// TwinCAT 3 PLC project TcPluginFramework
// Title: TcPluginFramework
// Company: Loupe
// ProjectVersion: 1.0.0
// ProgramVersion: 3.1.4024.0
// libraries:
//   Tc2_System, * (Beckhoff Automation GmbH)
//   TcUnit, * (www.tcunit.org)
// project tree:
//   DUTs/ ComponentBaseInternal.TcDUT, TaskBaseInternal.TcDUT
//   GVLs/ GVLPluginFramework.TcGVL
//   Interfaces/ IPlugin.TcIO, IPluginRunner.TcIO, ITaskState.TcIO
//   POUs/ ComponentBase.TcPOU, LogMessage.TcPOU, PluginRunner.TcPOU, TaskBase.TcPOU
//   Test/ TaskBaseExtended.TcPOU, TESTPRG.TcPOU

// ---- DUTs/ComponentBaseInternal.TcDUT
TYPE
    ComponentBaseInternal :
    STRUCT
        _initDone : BOOL;
        _ready : BOOL;
        _plugins : PluginRunner;
    END_STRUCT
END_TYPE

// ---- DUTs/TaskBaseInternal.TcDUT
TYPE
    TaskBaseInternal :
    STRUCT
        _state : UDINT;
        _newCommand : BOOL;
    END_STRUCT
END_TYPE

// ---- GVLs/GVLPluginFramework.TcGVL
{attribute 'qualified_only'}
VAR_GLOBAL
END_VAR
VAR_GLOBAL CONSTANT
	MAX_NUM_PLUGIN_RUNNERS: USINT := 20;
	MAI_NUM_PLUGIN_RUNNERS: USINT := MAX_NUM_PLUGIN_RUNNERS - 1;
END_VAR
VAR_GLOBAL
    LogLevel : INT;
END_VAR

// ---- Interfaces/IPlugin.TcIO
// Copyright (c) 2024 Loupe (https://loupe.team), provided under the MIT License.

INTERFACE IPlugin EXTENDS __SYSTEM.IQueryInterface

METHOD Run : BOOL
VAR_INPUT
END_VAR
END_METHOD

END_INTERFACE

// ---- Interfaces/IPluginRunner.TcIO
// Copyright (c) 2024 Loupe (https://loupe.team), provided under the MIT License.

INTERFACE IPluginRunner EXTENDS __System.IQueryInterface

METHOD RegisterPlugin
VAR_INPUT
    plugin : IPlugin;
END_VAR
END_METHOD

END_INTERFACE

// ---- Interfaces/ITaskState.TcIO
// Copyright (c) 2024 Loupe (https://loupe.team), provided under the MIT License.

INTERFACE ITaskState

METHOD Cyclic : BOOL
END_METHOD

METHOD Inihibits : BOOL
VAR_INPUT
END_VAR
END_METHOD

METHOD NewCommandState : BOOL
VAR_INPUT
    newTaskState : ENUM;
END_VAR
END_METHOD

PROPERTY NewTaskCommand : BOOL
GET
END_GET
END_PROPERTY

METHOD StateErrored : BOOL
VAR_INPUT
END_VAR
END_METHOD

METHOD StateFinished : BOOL
VAR_INPUT
END_VAR
END_METHOD

METHOD StateMachine : BOOL
VAR_INPUT
END_VAR
END_METHOD

{attribute 'monitoring' := 'call'}
PROPERTY TaskReady : Bool
GET
END_GET
SET
END_SET
END_PROPERTY

{attribute 'monitoring' := 'call'}
PROPERTY TaskState : ENUM
GET
END_GET
END_PROPERTY

METHOD UpdateState : BOOL
VAR_INPUT
END_VAR
END_METHOD

END_INTERFACE

// ---- POUs/ComponentBase.TcPOU
FUNCTION_BLOCK ABSTRACT ComponentBase IMPLEMENTS IPluginRunner, IPlugin
VAR
    _componentBase : ComponentBaseInternal;
END_VAR

// Copyright (c) 2024 Loupe (https://loupe.team), provided under the MIT License.

Run();

METHOD Cyclic : BOOL
// Copyright (c) 2024 Loupe (https://loupe.team), provided under the MIT License.

//This method is meant to be overridden to contain any cyclic function block calls
END_METHOD

METHOD Init : BOOL
VAR_INPUT
END_VAR
VAR
    nData : UDINT;
    pData : PVOID;
END_VAR
// Copyright (c) 2024 Loupe (https://loupe.team), provided under the MIT License.

InitComplete();
END_METHOD

METHOD InitComplete
VAR_INPUT
END_VAR
// Copyright (c) 2024 Loupe (https://loupe.team), provided under the MIT License.

_componentBase._initDone := TRUE;
LogMessage(0, 'Init Complete');
END_METHOD

METHOD RegisterPlugin
VAR_INPUT
    plugin : IPlugin;
END_VAR
// Copyright (c) 2024 Loupe (https://loupe.team), provided under the MIT License.

_componentBase._plugins.RegisterPlugin(plugin);
END_METHOD

METHOD Run : BOOL
VAR_INPUT
END_VAR
// Copyright (c) 2024 Loupe (https://loupe.team), provided under the MIT License.

//If we aren't initialized, call init
IF NOT _componentBase._initDone THEN

    //Init any derived classes
    THIS^.Init();

END_IF

runPlugins();

//Init() was successful, call cyclic
IF _componentBase._initDone THEN

    THIS^.Running();

END_IF
END_METHOD

METHOD Running : BOOL
VAR_INPUT
END_VAR
// Copyright (c) 2024 Loupe (https://loupe.team), provided under the MIT License.

// Run the main code
THIS^.Simulation();

THIS^.Cyclic();
END_METHOD

METHOD PRIVATE RunPlugins
// Copyright (c) 2024 Loupe (https://loupe.team), provided under the MIT License.

_componentBase._plugins.runPlugins();
END_METHOD

METHOD Simulation : BOOL
VAR_INPUT
END_VAR
// Copyright (c) 2024 Loupe (https://loupe.team), provided under the MIT License.
END_METHOD

END_FUNCTION_BLOCK

// ---- POUs/LogMessage.TcPOU
FUNCTION LogMessage
VAR_INPUT
    Level : INT;
    Message : STRING;
END_VAR

// Copyright (c) 2024 Loupe (https://loupe.team), provided under the MIT License.

IF Level >= GVLPluginFramework.LogLevel THEN
    ADSLOGSTR(msgCtrlMask := ADSLOG_MSGTYPE_LOG,
        msgFmtStr := Message,
        strArg := '');
END_IF

END_FUNCTION

// ---- POUs/PluginRunner.TcPOU
FUNCTION_BLOCK PluginRunner IMPLEMENTS IPluginRunner
VAR
    _plugins : ARRAY[0..GVLPluginFramework.MAI_NUM_PLUGIN_RUNNERS] OF IPlugin;
END_VAR

// Copyright (c) 2024 Loupe (https://loupe.team), provided under the MIT License.

METHOD RegisterPlugin
VAR_INPUT
    plugin : IPlugin;
END_VAR
VAR
    i : INT;
END_VAR
// Copyright (c) 2024 Loupe (https://loupe.team), provided under the MIT License.

FOR i := 0 TO (SIZEOF(_plugins) / SIZEOF(_plugins[0])) - 1 DO
    //We have a new slot
    IF _plugins[i] = 0 THEN
        _plugins[i] := plugin;
        RETURN;
        //We already added this plugin
    ELSIF _plugins[i] = plugin THEN
        RETURN;
    END_IF
END_FOR
END_METHOD

METHOD RunPlugins
VAR
    i : INT;
END_VAR
// Copyright (c) 2024 Loupe (https://loupe.team), provided under the MIT License.

FOR i := 0 TO (SIZEOF(_plugins) / SIZEOF(_plugins[0])) - 1 DO
    IF _plugins[i] <> 0 THEN
        _plugins[i].Run();
    ELSE
        EXIT;
    END_IF
END_FOR
END_METHOD

END_FUNCTION_BLOCK

// ---- POUs/TaskBase.TcPOU
FUNCTION_BLOCK ABSTRACT TaskBase EXTENDS ComponentBase IMPLEMENTS ITaskState
VAR
    _taskBase : TaskBaseInternal;
END_VAR

// Copyright (c) 2024 Loupe (https://loupe.team), provided under the MIT License.

METHOD Inihibits : BOOL
// Copyright (c) 2024 Loupe (https://loupe.team), provided under the MIT License.

//This method is meant to be overriden
END_METHOD

METHOD NewCommandState : BOOL
VAR_INPUT
    newTaskState : ENUM;
END_VAR
// Copyright (c) 2024 Loupe (https://loupe.team), provided under the MIT License.

_taskBase._newCommand := TRUE;
_taskBase._state := newTaskState;
END_METHOD

{warning 'add property implementation'}
PROPERTY NewTaskCommand : BOOL
GET
// Copyright (c) 2024 Loupe (https://loupe.team), provided under the MIT License.

// TODO implement
//newTaskCommand :=
END_GET
END_PROPERTY

METHOD Running : BOOL
VAR_INPUT
END_VAR
// Copyright (c) 2024 Loupe (https://loupe.team), provided under the MIT License.

THIS^.Simulation();

IF newTaskCommand THEN

    IF taskReady THEN

        THIS^.Inihibits();

        THIS^.UpdateState();

    ELSE

        //REJECTED		

    END_IF
END_IF

THIS^.StateMachine();

THIS^.Cyclic();
END_METHOD

METHOD StateErrored : BOOL
VAR_INPUT
END_VAR
// Copyright (c) 2024 Loupe (https://loupe.team), provided under the MIT License.
END_METHOD

METHOD StateFinished : BOOL
VAR_INPUT
END_VAR
// Copyright (c) 2024 Loupe (https://loupe.team), provided under the MIT License.

_taskBase._state := 0;
END_METHOD

METHOD StateMachine : BOOL
// Copyright (c) 2024 Loupe (https://loupe.team), provided under the MIT License.
END_METHOD

//Ready indicates that the task is ready to accept commands
{attribute 'monitoring' := 'call'}
PROPERTY TaskReady : BOOL
GET
// Copyright (c) 2024 Loupe (https://loupe.team), provided under the MIT License.

taskReady := _componentBase._ready;
END_GET
SET
// Copyright (c) 2024 Loupe (https://loupe.team), provided under the MIT License.

_componentBase._ready := taskReady;
END_SET
END_PROPERTY

//Gets the current state of the system
{attribute 'monitoring' := 'call'}
PROPERTY TaskState : ENUM
GET
// Copyright (c) 2024 Loupe (https://loupe.team), provided under the MIT License.

taskState := _taskBase._state;
END_GET
END_PROPERTY

METHOD UpdateState : BOOL
// Copyright (c) 2024 Loupe (https://loupe.team), provided under the MIT License.
END_METHOD

END_FUNCTION_BLOCK

// ---- Test/TaskBaseExtended.TcPOU
FUNCTION_BLOCK TaskBaseExtended EXTENDS TaskBase
VAR_INPUT
END_VAR
VAR_OUTPUT
END_VAR
VAR
END_VAR

END_FUNCTION_BLOCK

// ---- Test/TESTPRG.TcPOU
PROGRAM TESTPRG
VAR
	// Currently there are no tests, except instantiating FUBs to make sure they build
	base : ComponentBase;
	runner : PluginRunner;
	taskBaseExtended : TaskBase;
END_VAR

TcUnit.RUN();

END_PROGRAM
